FUNCTION_BLOCK MPC_LEVEL (* Basic FB with empty ECC *)
  (* Standard: 61499-2 *)
  (* Version 1.0, 2026-04-25, guilh *)
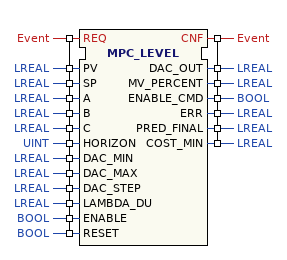
  EVENT_INPUT
    REQ WITH PV, SP, A, B, C, HORIZON, DAC_MIN, DAC_MAX, DAC_STEP, LAMBDA_DU, ENABLE, RESET;
  END_EVENT
  EVENT_OUTPUT
    CNF WITH DAC_OUT, MV_PERCENT, ENABLE_CMD, ERR, PRED_FINAL, COST_MIN;
  END_EVENT
  VAR_INPUT
    PV : LREAL;
    SP : LREAL;
    A : LREAL;
    B : LREAL;
    C : LREAL;
    HORIZON : UINT;
    DAC_MIN : LREAL;
    DAC_MAX : LREAL;
    DAC_STEP : LREAL;
    LAMBDA_DU : LREAL;
    ENABLE : BOOL;
    RESET : BOOL;
  END_VAR
  VAR_OUTPUT
    DAC_OUT : LREAL;
    MV_PERCENT : LREAL;
    ENABLE_CMD : BOOL;
    ERR : LREAL;
    PRED_FINAL : LREAL;
    COST_MIN : LREAL;
  END_VAR
  VAR
    last_dac : LREAL;
    best_dac : LREAL;
    best_cost : LREAL;
    dac_candidate : LREAL;
    y_pred : LREAL;
    pred_error : LREAL;
    delta_dac : LREAL;
    cost : LREAL;
    i : UINT;
    h : UINT;
  END_VAR
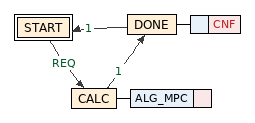
  EC_STATES
    START; (* Initial State *)
    CALC : ALG_MPC;
    DONE : -> CNF;
  END_STATES
  EC_TRANSITIONS
    START TO CALC := REQ;
    CALC TO DONE := 1;
    DONE TO START := 1;
  END_TRANSITIONS
  ALGORITHM ALG_MPC IN ST:
IF RESET THEN
    last_dac := 0.0;
END_IF;

ERR := SP - PV;

IF NOT ENABLE THEN
    DAC_OUT := 0.0;
    MV_PERCENT := 0.0;
    ENABLE_CMD := FALSE;
    PRED_FINAL := PV;
    COST_MIN := 0.0;
    last_dac := 0.0;

ELSE
    best_cost := 1.0E+30;
    best_dac := last_dac;
    PRED_FINAL := PV;

    IF HORIZON = 0 THEN
        h := 1;
    ELSE
        h := HORIZON;
    END_IF;

    dac_candidate := DAC_MIN;

    WHILE dac_candidate <= DAC_MAX DO

        y_pred := PV;
        cost := 0.0;

        i := 1;
        WHILE i <= h DO
            y_pred := A * y_pred + B * dac_candidate + C;
            pred_error := SP - y_pred;
            cost := cost + pred_error * pred_error;
            i := i + 1;
        END_WHILE;

        delta_dac := dac_candidate - last_dac;
        cost := cost + LAMBDA_DU * delta_dac * delta_dac;

        IF cost < best_cost THEN
            best_cost := cost;
            best_dac := dac_candidate;
            PRED_FINAL := y_pred;
        END_IF;

        IF DAC_STEP <= 0.0 THEN
            dac_candidate := DAC_MAX + 1.0;
        ELSE
            dac_candidate := dac_candidate + DAC_STEP;
        END_IF;

    END_WHILE;

    IF best_dac > DAC_MAX THEN
        best_dac := DAC_MAX;
    ELSIF best_dac < DAC_MIN THEN
        best_dac := DAC_MIN;
    END_IF;

    DAC_OUT := best_dac;

    IF DAC_MAX > 0.0 THEN
        MV_PERCENT := (DAC_OUT / DAC_MAX) * 100.0;
    ELSE
        MV_PERCENT := 0.0;
    END_IF;

    IF DAC_OUT > 1.0 THEN
        ENABLE_CMD := TRUE;
    ELSE
        ENABLE_CMD := FALSE;
    END_IF;

    COST_MIN := best_cost;
    last_dac := DAC_OUT;
END_IF;
  END_ALGORITHM
END_FUNCTION_BLOCK
